FUNCTION_BLOCK FB_Index
VAR_INPUT
	InitVal : INT := 0;
	IncVal : INT := 1;
	UpperLimit	:	INT := 1;
END_VAR
VAR_OUTPUT
	
END_VAR
VAR
	Val	:	INT := InitVal;
END_VAR

(* Index FB
A. Wallace 2016-9-3

Why doesn't beckhoff have this as a builtin type?
*)

;

METHOD PUBLIC IncVal : INT
VAR_INPUT
END_VAR
IncVal := THIS^.Val;
Inc();
END_METHOD

ACTION Dec:
Val := LIMIT(InitVal, Val - IncVal, UpperLimit);
END_ACTION

ACTION Inc:
Val := Val + IncVal;
IF Val >  UpperLimit THEN Val := InitVal; END_IF
END_ACTION

END_FUNCTION_BLOCK

(* stored: Version 1.1.0.1, ProductVersion 3.1.4018.5
   POU FB_Index: Id {ca8a34e3-bd4f-442e-9caf-17285b4f6fa2}, SpecialFunc None
   Method IncVal: Id {39565696-334a-4053-9d1a-5f11c00bc35c}
   Action Dec: Id {8c309ae9-b73a-4c3f-8e68-797f70101636}
   Action Inc: Id {dddba33c-25fc-4806-a697-b15b846415dc} *)
